{attribute addProperty BoxType "EL6201-0000-0017"}
{attribute addProperty Id "Slave_1A_DI0BIT10.1251Slave_1A_DI1BIT10.1252Slave_1A_DI2BIT10.1253Slave_1A_DI3BIT10.1254Slave_1B_DI0BIT10.1255Slave_1B_DI1BIT10.1256Slave_1B_DI2BIT10.1257Slave_1B_DI3BIT10.1258"}
{attribute addProperty CRC "1093278896"}
{attribute addProperty SizeInBites "8"}
{attribute addProperty SizeInBytes "1"}
TYPE Slave_1_Inputs_412A1CB0 :
STRUCT
	{attribute addProperty Name "Slave_1A_DI0"}
	Slave_1A_DI0 : BIT;
	{attribute addProperty Name "Slave_1A_DI1"}
	Slave_1A_DI1 : BIT;
	{attribute addProperty Name "Slave_1A_DI2"}
	Slave_1A_DI2 : BIT;
	{attribute addProperty Name "Slave_1A_DI3"}
	Slave_1A_DI3 : BIT;
	{attribute addProperty Name "Slave_1B_DI0"}
	Slave_1B_DI0 : BIT;
	{attribute addProperty Name "Slave_1B_DI1"}
	Slave_1B_DI1 : BIT;
	{attribute addProperty Name "Slave_1B_DI2"}
	Slave_1B_DI2 : BIT;
	{attribute addProperty Name "Slave_1B_DI3"}
	Slave_1B_DI3 : BIT;
END_STRUCT
END_TYPE

(* stored: Version 1.2.0.0, ProductVersion 3.1.4024.9
   DUT Slave_1_Inputs_412A1CB0: Id {572efb45-f6d7-4d69-9fa6-9f6a4f0bafc6} *)
